// TIA Portal V21 export
VAR_GLOBAL   // PLC tag table "KAllStazione"
END_VAR
VAR_GLOBAL CONSTANT   // user constants
   KALLStazione_ConflittoMultiDest : Int := 1;   // Sono state attivate troppe destinazioni contemporanee
   KALLStazione_AlmenoUnaDiagnosticaAttiva : Int := 2;   // Presente almeno una segnalazione nella vista diagnostica
   KALLStazione_TimeoutRun : Int := 3;   // Timeout partenza della stazione
END_VAR
